RoboDK station: pick_and_place.rdk

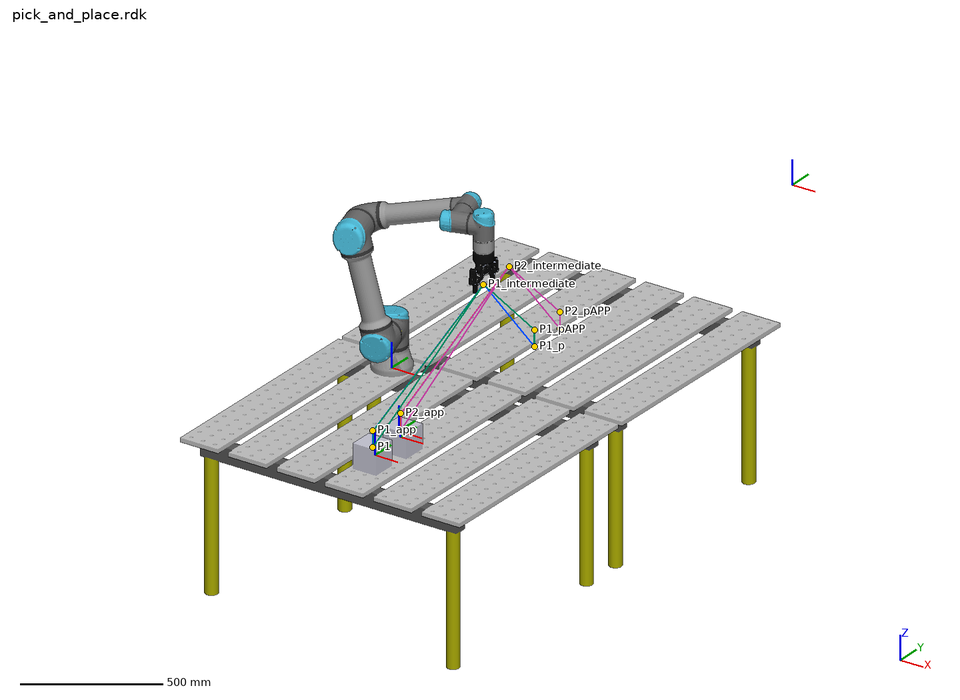
[picture v0: the station drawn from its stored meshes, robots at their saved joint values, targets as dots, program paths as lines]
Station P_and_P (saved by RoboDK 5.8.0). Poses are relative to the parent item; angles as X-Y-Z fixed-axis rotations.
  - frame Robot at (-310, 400, 0) mm
    - robot UR5e: 6 axes, payload 5 kg, reach 850 mm, repeatability 0.03 mm, weight 18.4 kg
        modified DH rows (alpha deg, a mm, theta deg, d mm): 0, 0, 0, 162.5; 90, 0, 180, 0; 0, 425, 0, 0; 0, 392.25, 0, 133.3; -90, 0, 0, 99.7; 90, 0, 180, 99.6
        joint limits [-360, -360, -360, -360, -360, -360] to [360, 360, 360, 360, 360, 360]; home [0, -90, -90, 0, 90, 0]; saved at [17.1, -76.424, -89.383, -104.193, 90, -162.9]
      - tool RobotiQ 2F-85 Gripper (Open), TCP at (0, 0, 130) mm, size 147.4 x 75 x 146.8 mm
  - frame World at (0, 0, 0) mm
    - object Tabel2 at (0, 990, 0) mm, size 1193.8 x 965.2 x 609.6 mm, geometry from Object Table.wrl
    - object Tabel1 at (0, 0, 0) mm, size 1193.8 x 965.2 x 609.6 mm, geometry from Object Table.wrl
  - frame Box1 at (100, -290, 50) mm
    - target P1 (Cartesian target) at (-7.39, -0.61, 27.2) mm, rotated rx 180 ry 0 rz 90 deg; joints [-50.16, -138.897, -61.25, -69.853, 90, -230.16] of UR5e
    - target P1_app (Cartesian target) at (-7.39, -0.61, 92.2) mm, rotated rx 180 ry 0 rz 90 deg; joints [-50.16, -136.009, -56.638, -77.353, 90, -230.16] of UR5e
    - target P1_intermediate (Cartesian target) at (-7.39, 674.39, 392.2) mm, rotated rx 180 ry 0 rz 90 deg; joints [17.1, -76.424, -89.383, -104.193, 90, -162.9] of UR5e
    - target P1_pAPP (Cartesian target) at (-7.39, 984.39, 92.2) mm, rotated rx 180 ry 0 rz 90 deg; joints [51.677, -96.929, -115.89, -57.181, 90, -128.323] of UR5e
    - target P1_p (Cartesian target) at (-7.39, 984.39, 27.2) mm, rotated rx 180 ry 0 rz 90 deg; joints [51.677, -103.067, -120.37, -46.563, 90, -128.323] of UR5e
  - frame Box2 at (90, -120, 50) mm
    - target P2_app (Cartesian target) at (2.61, -0.61, 92.2) mm, rotated rx 180 ry 0 rz 90 deg; joints [-49.606, -136.829, -55.16, -78.011, 90, -229.606] of UR5e
    - target P2 (Cartesian target) at (2.61, -0.61, 27.2) mm, rotated rx 180 ry 0 rz 90 deg; joints [-49.606, -139.648, -59.844, -70.508, 90, -229.606] of UR5e
    - target P2_intermediate (Cartesian target) at (-7.39, 674.39, 392.2) mm, rotated rx 180 ry 0 rz 90 deg; joints [39.887, -79.049, -87.381, -103.571, 90, -140.113] of UR5e
    - target P2_pAPP (Cartesian target) at (-7.39, 984.39, 92.2) mm, rotated rx 180 ry 0 rz 90 deg; joints [62.451, -110.614, -98.106, -61.28, 90, -117.549] of UR5e
    - target P2_p (Cartesian target) at (-7.39, 984.4, 27.2) mm, rotated rx 180 ry 0 rz 90 deg; joints [62.451, -115.484, -102.119, -52.397, 90, -117.549] of UR5e
  - frame Frame 6 at (0, 2400, 0) mm
  - program Attach (1 instructions, listed below)
  - program Detach (1 instructions, listed below)
  - program PP_box1 (12 instructions, listed below)
  - program PP_box2 (11 instructions, listed below)
  - program PPR_box1 (12 instructions, listed below)
  - program PPR_box2 (11 instructions, listed below)
  - program Main_pgm (4 instructions, listed below)
  - program Main_pgm(loop) (4 instructions, listed below)
  - object box2 at (100, -120, 50) mm, size 100 x 100 x 100 mm, geometry from box.sld
  - object box1 at (90, -290, 50) mm, size 100 x 100 x 100 mm, geometry from box.sld
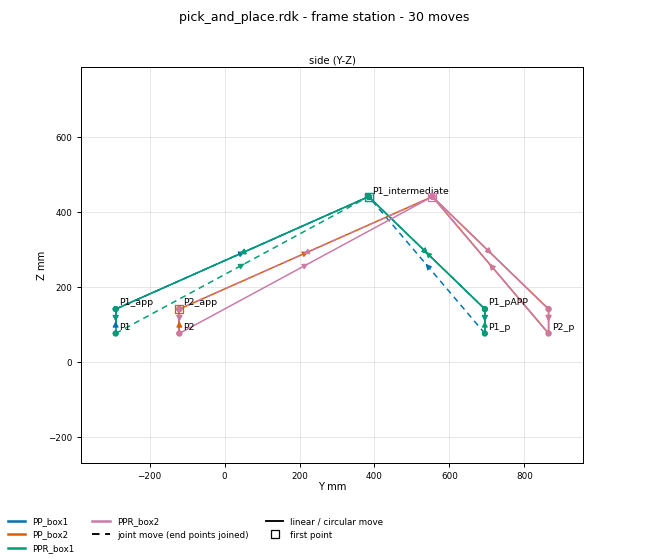
[picture p0: tool path of pick_and_place.rdk in frame station, 30 of 30 moves have a stored position in this frame; points joined in program order, loops and branches not executed]

--- program Attach (robot UR5e) ---
  Attach to RobotiQ 2F-85 Gripper (Open)

--- program Detach (robot UR5e) ---
  Detach from RobotiQ 2F-85 Gripper (Open)

--- program PP_box1 (robot UR5e) ---
  Set Ref.: Box1
  Set Tool: RobotiQ 2F-85 Gripper (Open)
  MoveJ (P1_intermediate)
  MoveL (P1_app)
  MoveJ (P1)
  Call Attach
  MoveL (P1_app)
  MoveJ (P1_intermediate)
  MoveL (P1_pAPP)
  MoveL (P1_p)
  Call Detach
  MoveJ (P1_intermediate)

--- program PP_box2 (robot UR5e) ---
  Set Ref.: Box2
  Set Tool: RobotiQ 2F-85 Gripper (Open)
  MoveJ (P2_app)
  MoveL (P2)
  Call Attach
  MoveJ (P2_app)
  MoveL (P2_intermediate)
  MoveL (P2_pAPP)
  MoveL (P2_p)
  Call Detach
  MoveL (P2_intermediate)

--- program PPR_box1 (robot UR5e) ---
  Set Ref.: Box1
  Set Tool: RobotiQ 2F-85 Gripper (Open)
  MoveJ (P1_intermediate)
  MoveL (P1_pAPP)
  MoveL (P1_p)
  Call Attach
  MoveL (P1_pAPP)
  MoveJ (P1_intermediate)
  MoveL (P1_app)
  MoveJ (P1)
  Call Detach
  MoveJ (P1_intermediate)

--- program PPR_box2 (robot UR5e) ---
  Set Ref.: Box2
  Set Tool: RobotiQ 2F-85 Gripper (Open)
  MoveL (P2_intermediate)
  MoveL (P2_pAPP)
  MoveL (P2_p)
  Call Attach
  MoveL (P2_intermediate)
  MoveJ (P2_app)
  MoveL (P2)
  Call Detach
  MoveL (P2_intermediate)

--- program Main_pgm (robot UR5e) ---
  Call PP_box1
  Call PP_box2
  Call PPR_box1
  Call PPR_box2

--- program Main_pgm(loop) (robot UR5e) ---
  Call PP_box1
  Call PP_box2
  Call PPR_box1
  Call PPR_box2
